ABB RobotStudio station: 6640_station_heavy_load.rsstn

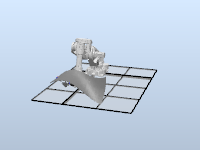
Station 6640_station_heavy_load (saved by RobotStudio 21.4.9700.0)
Controller IRB6640_180_255
  mechanical unit ROB_1: IRB6640_180_255__04_3, 6 joints, base frame (0, 0, 0) mm
Layout (positions relative to the parent item):
  - generic_fan_blade [part, from models\generic_fan_blade.rslib] at (2700, -800, 500) mm, rotated rx 90 ry 0 rz 90 deg
  - IRB6640_180_255__04_3 [mechanism, from Robots\IRB6640_180_255_G_04.rslib] at (0, 0, 0) mm; joint values [-0.0116, 1.1219, 0.1475, 0.7935, -1.6776, 2.9198] (rad or m)
  - HeavyTool [mechanism] at (1943.7, -164.29, 276.67) mm, rotated rx -0.46 ry -72.01 rz 131.64 deg
      TCP HeavyTool at (0, 0, 0) mm
      links: Paint gun
Attachment: HeavyTool is attached to IRB6640_180_255__04_3 / Link6
Targets, tools, work objects and paths stored in the station, written as RAPID:
! task T_ROB1
MODULE CalibData
  PERS tooldata MyNewTool:=[TRUE,[[50,0,450],[1,0,0,0]],[1,[0,0,1],[1,0,0,0],0,0,0]];
ENDMODULE

! task T_ROB1
MODULE CalibData
  PERS tooldata MyNewTool:=[TRUE,[[50,0,450],[1,0,0,0]],[1,[0,0,1],[1,0,0,0],0,0,0]];
ENDMODULE

! task T_ROB1
MODULE CalibData
  PERS tooldata MyNewTool:=[TRUE,[[50,0,450],[1,0,0,0]],[1,[0,0,1],[1,0,0,0],0,0,0]];
  PERS tooldata HeavyTool:=[TRUE,[[0,0,0],[1,0,0,0]],[100,[0,0,1],[1,0,0,0],0,0,0]];
ENDMODULE

